FUNCTION_BLOCK MockEvent IMPLEMENTS I_Event
VAR
	_name : T_MAXSTRING;
END_VAR

END_FUNCTION_BLOCK

(* stored: Version 1.1.0.1, ProductVersion 3.1.4024.12
   POU MockEvent: Id {2f9c554a-2034-412e-9e68-a68075e23a21}, SpecialFunc None *)
